// TIA Portal V19 export
VAR_GLOBAL   // PLC tag table "Unit2_Input"
END_VAR
